FUNCTION_BLOCK FB_VisionStation IMPLEMENTS I_ProcessEquipment
VAR
    // Commissioning FAIL/fault injection; a real camera FAIL cannot be overridden.
    // FALSE = use the real camera verdicts (default)
    // TRUE  = inject FAIL after valid camera evaluation
    bSimulatedFail              : BOOL := FALSE;
    bSimulatedFault             : BOOL := FALSE;

    bEnableInternal             : BOOL;
    bCommissionedInternal       : BOOL;
    bSafetyOkInternal           : BOOL;
    bSupervisionEnableInternal  : BOOL;

    // Nest support and intermediate stop removed from the mechanical design.


    // Vision / flipping tooling feedback.
    bHorizontalBackInternal     : BOOL;
    bHorizontalFrontInternal    : BOOL;
    bVerticalUpInternal         : BOOL;
    bVerticalDownInternal       : BOOL;

    bGripOpenedInternal         : BOOL;
    bGripClosedInternal         : BOOL;
    bRotate0Internal            : BOOL;
    bRotate180Internal          : BOOL;
    bRotate0RawInternal : BOOL;
    bRotate180RawInternal : BOOL;
    bCameraTriggerAcceptedInternal : BOOL;
    bCameraReadyForFlipInternal : BOOL;
    bUseOptimizedSequenceTimingInternal : BOOL;
    rtRotate0Raw : R_TRIG;
    tonFlipDeparture : TON;
    tFlipDepartureFilter : TIME := T#20MS;
    bFlipCaptureActive : BOOL;
    bFlipCaptureActivePrevious : BOOL;
    bFlipStart0Confirmed : BOOL;
    bFlipLeft0 : BOOL;
    bFlip90Seen : BOOL;
    bFlipTriggerLatched : BOOL;
    bFlipCaptureAccepted : BOOL;
    bFlipCaptureWindowMissed : BOOL;
	// Vision / Camera
	

    eStateInternal              : E_PatchStationState := E_PatchStationState.Disabled;
    usiStepInternal             : USINT := 0;
    bHomeInternal               : BOOL;
    bReadyInternal              : BOOL;
    bBusyInternal               : BOOL;
    bCompleteInternal           : BOOL;
    bFaultInternal              : BOOL;
    sDiagnosticInternal         : STRING(120);

    // Output requests.

    bHorizontalBackRequestInternal  : BOOL;
    bHorizontalFrontRequestInternal : BOOL;
    bVerticalUpRequestInternal      : BOOL;
    bVerticalDownRequestInternal    : BOOL;

    bGripCloseRequestInternal       : BOOL;
    bGripOpenRequestInternal        : BOOL;
    bRotate0RequestInternal         : BOOL;
    bRotate180RequestInternal       : BOOL;
	
	bTriggerRequestInternal			: BOOL;
	bChangeProgramRequestInternal	: BOOL;
	bGetResultsRequestInternal		: BOOL;
	bResetResultsRequestInternal	: BOOL;
	nSetProgramNumberInternal		: UDINT;
	bAcknowledgeResultsInternal		: BOOL;
	
	nCurrentProgramNumberInternal	: UDINT;
	bCameraResultsReadyInternal		: BOOL;
	nVisionResultsInternal			: ST_VisionResults;

    bStopRequestInternal        : BOOL;


    // Commissioning timing.
    tonStepDelay                : TON;
    tonRotate180Hold            : TON;
    tonMoveTimeout              : TON;

    tonToolingSensorConflict    : TON;

	tonChangeProgram			: TON := (PT := T#1S);

    tStepDelay                  : TIME := T#100MS;
    tRotate180Hold              : TIME := T#1S;
    tMoveTimeout                : TIME := T#30S;

    tToolingSensorConflict      : TIME := T#300MS;

	tTakingPictureWHileRotating	: TIME := T#100MS; // Delay AFTER the latched 90-degree marker; commission for the desired image.
	tDelayInspectionPlaceHolder	: TIME;

    bStepTargetReached          : BOOL;
    bToolingSensorConflict      : BOOL;
	
	rTrigger						: R_TRIG;
	tonCamera110Rearm             : TON;
	tonCameraTriggerDelay			: ARRAY [1..2] OF TON;
	tonTakingPictureWHileRotating	: TON;
	tonDelayInspectionPlaceHolder	: TON;

    stEmptyVisionResults        : ST_VisionResults;
    stResultInternal            : ST_ProcessResult;
    stProcessSettingsInternal : ST_CameraProcessSettings;
END_VAR

METHOD PUBLIC Cyclic
VAR_INPUT
END_VAR
VAR
	
	

END_VAR
tTakingPictureWHileRotating := UDINT_TO_TIME(stProcessSettingsInternal.udiMovingTriggerDelayMs);
// Marker tracking uses raw feedback; endpoint qualification is independent.
rtRotate0Raw(CLK := bRotate0RawInternal);
bFlipCaptureActive := bEnableInternal AND bCommissionedInternal AND bSafetyOkInternal
    AND NOT bStopRequestInternal
    AND (eStateInternal = E_PatchStationState.Processing) AND (usiStepInternal = 100);
IF NOT bFlipCaptureActive THEN
    bFlipStart0Confirmed := FALSE;
    bFlipLeft0 := FALSE;
    bFlip90Seen := FALSE;
    bFlipTriggerLatched := FALSE;
    bFlipCaptureAccepted := FALSE;
    bFlipCaptureWindowMissed := FALSE;
ELSIF NOT bFlipCaptureActivePrevious THEN
    bFlipStart0Confirmed := bRotate0Internal AND NOT bRotate180RawInternal;
    bFlipLeft0 := FALSE;
    bFlip90Seen := FALSE;
    bFlipTriggerLatched := FALSE;
    bFlipCaptureAccepted := FALSE;
    bFlipCaptureWindowMissed := NOT bFlipStart0Confirmed;
END_IF
tonFlipDeparture(IN := bFlipCaptureActive AND bFlipStart0Confirmed AND NOT bFlipLeft0
    AND NOT bRotate0RawInternal AND NOT bRotate180RawInternal, PT := tFlipDepartureFilter);
IF tonFlipDeparture.Q THEN bFlipLeft0 := TRUE; END_IF
IF bFlipCaptureActive AND bFlipLeft0 AND rtRotate0Raw.Q
    AND NOT bFlip90Seen AND NOT bRotate180RawInternal THEN
    bFlip90Seen := TRUE;
END_IF
tonTakingPictureWHileRotating(IN := bFlipCaptureActive AND bFlip90Seen,
    PT := tTakingPictureWHileRotating);
IF bFlipCaptureActive THEN
    IF bFlipTriggerLatched AND bCameraTriggerAcceptedInternal THEN bFlipCaptureAccepted := TRUE; END_IF
    IF bRotate180RawInternal AND NOT bFlipCaptureAccepted THEN
        bFlipCaptureWindowMissed := TRUE;
    ELSIF tonTakingPictureWHileRotating.Q AND NOT bFlipTriggerLatched
        AND NOT bFlipCaptureWindowMissed THEN
        IF nCurrentProgramNumberInternal = 1 THEN
            bFlipTriggerLatched := TRUE;
        ELSE
            bFlipCaptureWindowMissed := TRUE;
        END_IF
    END_IF
END_IF
bFlipCaptureActivePrevious := bFlipCaptureActive;

// Rearm inspection 2 after entry and confirmed program selection.
tonCamera110Rearm(
    IN := (eStateInternal = E_PatchStationState.Processing)
        AND (usiStepInternal = 110)
        AND (nCurrentProgramNumberInternal = 2)
        AND NOT tonCameraTriggerDelay[1].IN
        AND NOT tonCameraTriggerDelay[2].IN,
    PT := T#500MS
);

bTriggerRequestInternal :=
    (eStateInternal = E_PatchStationState.Processing)
    AND (
        ((usiStepInternal = 100) AND (nCurrentProgramNumberInternal = 1)
            AND bFlipTriggerLatched AND NOT bFlipCaptureWindowMissed)
        OR ((usiStepInternal = 10) AND (nCurrentProgramNumberInternal = 0)
            AND NOT tonCameraTriggerDelay[2].IN)
        OR ((usiStepInternal = 110) AND tonCamera110Rearm.Q)
        OR ((usiStepInternal = 180) AND (nCurrentProgramNumberInternal = 3))
    );
bGetResultsRequestInternal := FALSE;
bAcknowledgeResultsInternal := FALSE;
bChangeProgramRequestInternal := FALSE;
tonCameraTriggerDelay[1](PT := T#500MS);
// Keep the program 0-to-1 timer running while pick and mounting proceed.
IF (eStateInternal = E_PatchStationState.Processing)
    AND ((usiStepInternal = 10) OR (bUseOptimizedSequenceTimingInternal AND (usiStepInternal <= 90))) THEN
    tonCameraTriggerDelay[2](PT := T#200MS);
ELSE
    tonCameraTriggerDelay[2](PT := T#500MS);
END_IF
tonDelayInspectionPlaceHolder(PT := tDelayInspectionPlaceHolder);

 // ============================================================================
 // Vision Station / Flipping sequence
 // ============================================================================
 // Home:
 //
 // Process (active mechanical steps and camera inspections):
 //
 //   10  1st Vision Inspection - Program 0
 //   30  Vertical FULL DOWN - pick
 //   40  Grip CLOSE
 //   50  Vertical UP
 //   60  Horizontal FRONT
 //   80  Vertical UP before flip
 //   100  Rotate 180; timed Program 1 capture and result acquisition
 //   110  3rd Vision Inspection - Program 2
 //  150  Grip OPEN - release part
 //  160  Vertical UP after release
 //  170  Return tooling HOME
 //  180  4th Vision Inspection - Program 3
 //  190  Aggregate four camera verdicts, then Complete


// ============================================================================
// DEFAULT REQUESTS
// ============================================================================

// Default all requests OFF. Each active state below explicitly builds the
// desired command state and never energises opposing coils simultaneously.

bHorizontalBackRequestInternal := FALSE;
bHorizontalFrontRequestInternal := FALSE;
bVerticalUpRequestInternal := FALSE;
bVerticalDownRequestInternal := FALSE;

bGripCloseRequestInternal := FALSE;
bGripOpenRequestInternal := FALSE;
bRotate0RequestInternal := FALSE;
bRotate180RequestInternal := FALSE;

//bStepTargetReached := FALSE;
bFaultInternal := FALSE;


// ============================================================================
// HOME FEEDBACK
// ============================================================================

bHomeInternal :=
    bHorizontalBackInternal AND NOT bHorizontalFrontInternal
    AND bVerticalUpInternal AND NOT bVerticalDownInternal
    AND bGripOpenedInternal AND NOT bGripClosedInternal
    AND bRotate0Internal AND NOT bRotate180Internal;


// ============================================================================
// TOOLING SENSOR PLAUSIBILITY
// ============================================================================

bToolingSensorConflict :=
    (bHorizontalBackInternal AND bHorizontalFrontInternal)
    OR (bVerticalUpInternal AND bVerticalDownInternal)
    OR (bGripOpenedInternal AND bGripClosedInternal)
    OR (bRotate0RawInternal AND bRotate180RawInternal);

// End-position sensors can overlap briefly during pneumatic transitions.
// Only treat contradictory feedback as a real fault when it persists.
tonToolingSensorConflict(
    IN := bSupervisionEnableInternal
        AND bSafetyOkInternal
        AND bToolingSensorConflict,
    PT := tToolingSensorConflict
);


// ============================================================================
// MAIN STATE CONTROL
// ============================================================================

IF bEnableInternal AND bSimulatedFault THEN

    eStateInternal := E_PatchStationState.Fault;
    usiStepInternal := 0;
    sDiagnosticInternal := 'Vision: simulated station fault';


ELSIF bFlipCaptureWindowMissed THEN
    eStateInternal := E_PatchStationState.Fault;
    usiStepInternal := 0;
    bTriggerRequestInternal := FALSE;
    sDiagnosticInternal := 'Vision: rotation reference or moving-image window missed';
    stResultInternal.bValid := TRUE;
    stResultInternal.bPassed := FALSE;
    stResultInternal.eCode := E_ProcessResultCode.Fail;
    stResultInternal.udiFaultCode := 12;
    stResultInternal.udiAlertCode := 0;
    stResultInternal.sDetail := sDiagnosticInternal;

ELSIF tonToolingSensorConflict.Q THEN

    eStateInternal := E_PatchStationState.Fault;
    usiStepInternal := 0;
    sDiagnosticInternal := 'Vision: contradictory tooling sensors';


ELSIF bFaultInternal THEN

    // Fault state handled below.


ELSIF bStopRequestInternal THEN

    // Controlled station stop: start one deterministic return-to-home sequence.
    // Clear the request here so the homing step counter is not reset every scan.
    eStateInternal := E_PatchStationState.Homing;
    usiStepInternal := 0;
    bStopRequestInternal := FALSE;


ELSIF NOT bCommissionedInternal THEN

    eStateInternal := E_PatchStationState.Disabled;
    usiStepInternal := 0;
    sDiagnosticInternal := 'Vision: station disabled';


ELSIF NOT bSafetyOkInternal THEN

    eStateInternal := E_PatchStationState.Disabled;
    usiStepInternal := 0;
    sDiagnosticInternal := 'Vision: disabled by Safety';


ELSIF NOT bEnableInternal THEN

    IF bHomeInternal THEN

        eStateInternal := E_PatchStationState.Disabled;
        usiStepInternal := 0;
        sDiagnosticInternal := 'Vision: disabled - tooling home';

    ELSE

        eStateInternal := E_PatchStationState.Homing;
        usiStepInternal := 0;
        sDiagnosticInternal := 'Vision: disabled - returning tooling home';

    END_IF


ELSE

    CASE eStateInternal OF


        // ====================================================================
        // DISABLED / HOMING
        // ====================================================================

        E_PatchStationState.Disabled,
        E_PatchStationState.Homing:

            // Deterministic / collision-conscious home sequence used by
            // System Initialising and controlled station recovery.
            //
			// Defined HOME:

            // Request program 0 during homing; mechanical Ready still does not confirm camera Ready.
            
			//Leaving camera with the right program to performance first test--------------------------
			
			IF nCurrentProgramNumberInternal<> 0 THEN
				
				nSetProgramNumberInternal				:= 0;
				bChangeProgramRequestInternal			:= TRUE;
				
			ELSIF nCurrentProgramNumberInternal = 0 THEN
				
				bChangeProgramRequestInternal			:= FALSE;
				
			END_IF
			

            
			//-------------------------------------------------------------------------------------------
            IF usiStepInternal = 0 THEN

                IF bHomeInternal THEN
                    usiStepInternal := 70;
                ELSE
                    usiStepInternal := 10;
                END_IF

            END_IF


            CASE usiStepInternal OF
			

				10: // Vertical UP

                    bVerticalUpRequestInternal := NOT bVerticalUpInternal;

                    bStepTargetReached :=
                        bVerticalUpInternal
                        AND NOT bVerticalDownInternal;

                    sDiagnosticInternal := 'Vision homing: vertical UP';


                30: // Rotate gripper to 0 deg

                    bVerticalUpRequestInternal := NOT bVerticalUpInternal;

                    bRotate0RequestInternal := NOT bRotate0Internal;

                    bStepTargetReached :=
                        bRotate0Internal
                        AND NOT bRotate180Internal;

                    sDiagnosticInternal := 'Vision homing: rotate grip to 0 deg';


                40: // Grip OPEN

                    bVerticalUpRequestInternal := NOT bVerticalUpInternal;

                    bRotate0RequestInternal := NOT bRotate0Internal;
                    bGripOpenRequestInternal := NOT bGripOpenedInternal;

                    bStepTargetReached :=
                        bGripOpenedInternal
                        AND NOT bGripClosedInternal;

                    sDiagnosticInternal := 'Vision homing: grip OPEN';


                60: // Horizontal slide BACK

                    bVerticalUpRequestInternal := NOT bVerticalUpInternal;

                    bRotate0RequestInternal := NOT bRotate0Internal;
                    bGripOpenRequestInternal := NOT bGripOpenedInternal;



                    bHorizontalBackRequestInternal := NOT bHorizontalBackInternal;

                    bStepTargetReached :=
                        bHorizontalBackInternal
                        AND NOT bHorizontalFrontInternal;

                    sDiagnosticInternal := 'Vision homing: horizontal slide BACK';


                70: // Verify complete HOME before declaring Ready

                    bHorizontalBackRequestInternal := NOT bHorizontalBackInternal;
                    bVerticalUpRequestInternal := NOT bVerticalUpInternal;



                    bGripOpenRequestInternal := NOT bGripOpenedInternal;
                    bRotate0RequestInternal := NOT bRotate0Internal;

                    // Modified by Thays - TEMPORARY: verify mechanical HOME without requiring Keyence program 0.
                    // bStepTargetReached := bHomeInternal AND (nCurrentProgramNumberInternal = 0);
                    bStepTargetReached := bHomeInternal;

                    sDiagnosticInternal := 'Vision homing: verifying HOME';
					

                ELSE

                    usiStepInternal := 10;
                    bStepTargetReached := FALSE;

            END_CASE


            tonStepDelay(
                IN := bStepTargetReached,
                PT := tStepDelay
            );

            tonMoveTimeout(
                IN := NOT bStepTargetReached,
                PT := tMoveTimeout
            );


            // ================================================================
            // HOMING TIMEOUT SUPERVISION
            // ================================================================

            IF tonMoveTimeout.Q THEN

                tonMoveTimeout(IN := FALSE);
                tonStepDelay(IN := FALSE);

                eStateInternal := E_PatchStationState.Fault;
                usiStepInternal := 0;

                sDiagnosticInternal := 'Vision: homing movement timeout';

                stResultInternal.bValid := TRUE;
                stResultInternal.bPassed := FALSE;
                stResultInternal.eCode := E_ProcessResultCode.Fail;
                stResultInternal.udiFaultCode := 11;
                stResultInternal.udiAlertCode := 0;
                stResultInternal.sDetail := 'Vision homing movement timeout';


            ELSIF tonStepDelay.Q THEN

                tonMoveTimeout(IN := FALSE);
                tonStepDelay(IN := FALSE);

                IF usiStepInternal < 70 THEN

                    IF usiStepInternal = 10 THEN
                        usiStepInternal := 30;
                    ELSIF usiStepInternal = 40 THEN
                        usiStepInternal := 60;
                    ELSE
                        usiStepInternal := usiStepInternal + 10;
                    END_IF

                ELSE

                    eStateInternal := E_PatchStationState.Ready;
                    usiStepInternal := 0;
                    sDiagnosticInternal := 'Vision: ready - tooling home';
					bStepTargetReached					:= FALSE;

                END_IF

            END_IF


        // ====================================================================
        // READY
        // ====================================================================

        E_PatchStationState.Ready:

            // Reset can enter Ready directly when tooling is already home.
            // Restore the camera independently of the mechanical homing path.
            IF nCurrentProgramNumberInternal <> 0 THEN
                nSetProgramNumberInternal := 0;
                bChangeProgramRequestInternal := TRUE;
            END_IF

            tonStepDelay(IN := FALSE);
            tonRotate180Hold(IN := FALSE);
            tonMoveTimeout(IN := FALSE);

            // Hold/restore the defined HOME position.

            bHorizontalBackRequestInternal := NOT bHorizontalBackInternal;
            bVerticalUpRequestInternal := NOT bVerticalUpInternal;



            bGripOpenRequestInternal := NOT bGripOpenedInternal;
            bRotate0RequestInternal := NOT bRotate0Internal;

            IF NOT bHomeInternal THEN

                eStateInternal := E_PatchStationState.Homing;
                sDiagnosticInternal := 'Vision: lost home - recovering';

            ELSE

                sDiagnosticInternal := 'Vision: ready - waiting for cycle start';

            END_IF


        // ====================================================================
        // PROCESSING
        // ====================================================================

        E_PatchStationState.Processing:

            // Each scan must prove completion of the active step.
            bStepTargetReached := FALSE;

            // Continue the first camera handshake while automatic tooling moves.
            IF (usiStepInternal = 10) OR (bUseOptimizedSequenceTimingInternal AND (usiStepInternal <= 90)) THEN
                IF tonCameraTriggerDelay[1].Q THEN
                    tonCameraTriggerDelay[1].IN := FALSE;
                    tonCameraTriggerDelay[2].IN := TRUE;
                END_IF

                IF tonCameraTriggerDelay[2].IN THEN
                    nSetProgramNumberInternal := 1;
                    bChangeProgramRequestInternal := (nCurrentProgramNumberInternal <> 1);
                ELSIF (usiStepInternal = 10) AND (nCurrentProgramNumberInternal = 0)
                    AND bCameraResultsReadyInternal THEN
                    bGetResultsRequestInternal := TRUE;
                    bAcknowledgeResultsInternal := TRUE;
                    tonCameraTriggerDelay[1].IN := TRUE;
                ELSIF (usiStepInternal = 10) AND NOT tonCameraTriggerDelay[1].IN
                    AND (nCurrentProgramNumberInternal <> 0) THEN
                    nSetProgramNumberInternal := 0;
                    bChangeProgramRequestInternal := TRUE;
                END_IF
            END_IF

            CASE usiStepInternal OF

                10: // Keep the part stationary until the first result has been copied.
                    bStepTargetReached := nVisionResultsInternal.aInspectionCompleted[1]
                        AND (tonCameraTriggerDelay[1].IN OR tonCameraTriggerDelay[2].IN)
                        AND (bUseOptimizedSequenceTimingInternal
                            OR (tonCameraTriggerDelay[2].Q AND (nCurrentProgramNumberInternal = 1)));
                    sDiagnosticInternal := 'Vision: Camera first inspection';

                20: // Prepare existing tooling for pick.
                    bHorizontalBackRequestInternal := NOT bHorizontalBackInternal;
                    bVerticalUpRequestInternal := NOT bVerticalUpInternal;
                    bGripOpenRequestInternal := NOT bGripOpenedInternal;
                    bRotate0RequestInternal := NOT bRotate0Internal;
                    bStepTargetReached := bHorizontalBackInternal AND NOT bHorizontalFrontInternal
                        AND bVerticalUpInternal AND NOT bVerticalDownInternal
                        AND bGripOpenedInternal AND NOT bGripClosedInternal
                        AND bRotate0Internal AND NOT bRotate180Internal;
                    sDiagnosticInternal := 'Vision: preparing pick tooling';

                30:

                    bHorizontalBackRequestInternal := NOT bHorizontalBackInternal;

                    // Coil5 = OFF.


                    bVerticalDownRequestInternal := NOT bVerticalDownInternal;

                    bGripOpenRequestInternal := NOT bGripOpenedInternal;
                    bRotate0RequestInternal := NOT bRotate0Internal;

                    bStepTargetReached :=
                        bVerticalDownInternal
                        AND NOT bVerticalUpInternal;

                    sDiagnosticInternal := 'Vision: vertical FULL DOWN - pick';


                // ------------------------------------------------------------
                // STEP 40 - GRIP CLOSE AT FULL DOWN
                // ------------------------------------------------------------

                40:

                    bHorizontalBackRequestInternal := NOT bHorizontalBackInternal;

                    // Keep stop retracted while gripping at FULL DOWN.


                    bVerticalDownRequestInternal := NOT bVerticalDownInternal;

                    bGripCloseRequestInternal := NOT bGripClosedInternal;
                    bRotate0RequestInternal := NOT bRotate0Internal;

                    bStepTargetReached :=
                        bGripClosedInternal
                        AND NOT bGripOpenedInternal;

                    sDiagnosticInternal := 'Vision: grip CLOSE at full DOWN';


                // ------------------------------------------------------------
                // STEP 50 - VERTICAL UP
                // ------------------------------------------------------------

                50:

                    bHorizontalBackRequestInternal := NOT bHorizontalBackInternal;
                    bVerticalUpRequestInternal := NOT bVerticalUpInternal;

                    // Keep stop retracted until vertical is safely UP.


                    bGripCloseRequestInternal := NOT bGripClosedInternal;
                    bRotate0RequestInternal := NOT bRotate0Internal;

                    bStepTargetReached :=
                        bVerticalUpInternal
                        AND NOT bVerticalDownInternal;

                    sDiagnosticInternal := 'Vision: vertical UP with part';


                // ------------------------------------------------------------
                // STEP 60 - HORIZONTAL FRONT
                // ------------------------------------------------------------

                60:

                    bHorizontalFrontRequestInternal := NOT bHorizontalFrontInternal;
                    bVerticalUpRequestInternal := NOT bVerticalUpInternal;

                    // before commanding the next DOWN movement.


                    bGripCloseRequestInternal := NOT bGripClosedInternal;
                    bRotate0RequestInternal := NOT bRotate0Internal;

                    bStepTargetReached :=
                        bHorizontalFrontInternal
                        AND NOT bHorizontalBackInternal;

                    sDiagnosticInternal := 'Vision: horizontal FRONT';


                // ------------------------------------------------------------
                // ------------------------------------------------------------

                70: // Two-position vertical cylinder: use actual DOWN feedback.
                    bHorizontalFrontRequestInternal := NOT bHorizontalFrontInternal;
                    bVerticalDownRequestInternal := NOT bVerticalDownInternal;
                    bGripCloseRequestInternal := NOT bGripClosedInternal;
                    bRotate0RequestInternal := NOT bRotate0Internal;
                    bStepTargetReached := bVerticalDownInternal AND NOT bVerticalUpInternal;
                    IF bStepTargetReached THEN
                        sDiagnosticInternal := 'Vision: PBUP mounting - holding DOWN for 1 s';
                    ELSE
                        sDiagnosticInternal := 'Vision: vertical DOWN - front position';
                    END_IF

                80:

                    bHorizontalFrontRequestInternal := NOT bHorizontalFrontInternal;
                    bVerticalUpRequestInternal := NOT bVerticalUpInternal;



                    bGripCloseRequestInternal := NOT bGripClosedInternal;
                    bRotate0RequestInternal := NOT bRotate0Internal;

                    // FIX: removed simultaneous retract request from Step 70.
                    // OLD: bStepTargetReached :=
                    //          (bVerticalUpInternal AND NOT bVerticalDownInternal)
                    bStepTargetReached :=
                        bVerticalUpInternal
                        AND NOT bVerticalDownInternal;

                    sDiagnosticInternal := 'Vision: vertical UP before flip';

                // ------------------------------------------------------------
                // ------------------------------------------------------------

                90: // Verify clearance before rotation; no nest support is fitted.
                    bHorizontalFrontRequestInternal := NOT bHorizontalFrontInternal;
                    bVerticalUpRequestInternal := NOT bVerticalUpInternal;
                    bGripCloseRequestInternal := NOT bGripClosedInternal;
                    bRotate0RequestInternal := NOT bRotate0Internal;
                    bStepTargetReached := bVerticalUpInternal AND NOT bVerticalDownInternal
                        AND bRotate0Internal AND NOT bRotate180Internal;
                    IF bUseOptimizedSequenceTimingInternal
                        AND NOT (tonCameraTriggerDelay[2].Q AND (nCurrentProgramNumberInternal = 1)
                            AND bCameraReadyForFlipInternal) THEN
                        bStepTargetReached := FALSE;
                        sDiagnosticInternal := 'Vision: waiting for camera program 1 ready';
                    ELSE
                        sDiagnosticInternal := 'Vision: verify UP before flip';
                    END_IF

                100: // Support retraction was confirmed in step 90.

					// Program 1 trigger now follows the first valid 90-degree marker.

                    bHorizontalFrontRequestInternal := NOT bHorizontalFrontInternal;
                    bVerticalUpRequestInternal := NOT bVerticalUpInternal;


                    bGripCloseRequestInternal := NOT bGripClosedInternal;
                    bRotate180RequestInternal := NOT bRotate180Internal;

                    // Acquire program 1 before requesting program 2.
                    
					//Camera
					IF nCurrentProgramNumberInternal = 1 THEN
					
					IF bCameraResultsReadyInternal AND NOT tonCameraTriggerDelay[2].IN THEN
						
						bGetResultsRequestInternal			:= TRUE;
						bAcknowledgeResultsInternal			:= TRUE;
						tonCameraTriggerDelay[1].IN			:= TRUE;
						
						
					END_IF
					
					END_IF
					IF tonCameraTriggerDelay[1].Q THEN
							
							bGetResultsRequestInternal			:= FALSE;
							bAcknowledgeResultsInternal			:= FALSE;
							nSetProgramNumberInternal			:= 2;
							tonDelayInspectionPlaceHolder.IN	:= TRUE;
							bChangeProgramRequestInternal		:= TRUE;
							tonCameraTriggerDelay[2].IN			:= TRUE;
							tonCameraTriggerDelay[1].IN			:= FALSE;
							
							
					END_IF
					// Hold program selection until the camera reports the requested program.
                    IF tonCameraTriggerDelay[2].IN THEN
                        nSetProgramNumberInternal := 2;
                        bChangeProgramRequestInternal := (nCurrentProgramNumberInternal <> 2);
                    END_IF
                    IF tonCameraTriggerDelay[2].Q AND (nCurrentProgramNumberInternal = 2) THEN
							
							
							bChangeProgramRequestInternal		:= FALSE;

							
							
					END_IF
					// The moving-image delay is not restarted by the program-change placeholder.
					
					bStepTargetReached := tonDelayInspectionPlaceHolder.Q
                        AND (nCurrentProgramNumberInternal = 2)
                        AND bRotate180Internal AND NOT bRotate0Internal;
					
					                    
                    // Physical 180 completion is now qualified above before inspection 3.
                    //tonDelayInspectionPlaceHolder.IN := bRotate180Internal AND NOT bRotate0Internal;
                    //bStepTargetReached := bRotate180Internal AND NOT bRotate0Internal AND tonDelayInspectionPlaceHolder.Q;
                    sDiagnosticInternal := 'Vision: rotate 180, marker-based image 2';
				
                // Pending: accepted-trigger/fresh-result handshake and supervised visual inspection recovery.
        
				// ------------------------------------------------------------
                // STEP 110 - CAMERA PROGRAM 2 - THIRD INSPECTION
                // ------------------------------------------------------------
				
				110:
					tonDelayInspectionPlaceHolder.IN		:= FALSE;

                    // Acquire program 2 before requesting program 3.
                    
					IF nCurrentProgramNumberInternal = 2 THEN
					
					IF bCameraResultsReadyInternal AND NOT tonCameraTriggerDelay[2].IN THEN
						
						bGetResultsRequestInternal			:= TRUE;
						bAcknowledgeResultsInternal			:= TRUE;
						tonCameraTriggerDelay[1].IN			:= TRUE;
						
						
					END_IF
					END_IF
					
					IF tonCameraTriggerDelay[1].Q THEN
							
							bGetResultsRequestInternal			:= FALSE;
							bAcknowledgeResultsInternal			:= FALSE;
							nSetProgramNumberInternal			:= 3;
							bChangeProgramRequestInternal		:= TRUE;
							tonCameraTriggerDelay[2].IN			:= TRUE;
							tonCameraTriggerDelay[1].IN			:= FALSE;
							
							
					END_IF
					// Hold program selection until the camera reports the requested program.
                    IF tonCameraTriggerDelay[2].IN THEN
                        nSetProgramNumberInternal := 3;
                        bChangeProgramRequestInternal := (nCurrentProgramNumberInternal <> 3);
                    END_IF
                    IF tonCameraTriggerDelay[2].Q AND (nCurrentProgramNumberInternal = 3) THEN
							
							
							bChangeProgramRequestInternal		:= FALSE;
							bStepTargetReached					:= TRUE;
                            // Keep delay 2 complete until this step advances.
							
							
					END_IF
				
                    
                    //bStepTargetReached := TRUE; // Modified by Thays - no camera inspection result.

                // ------------------------------------------------------------
                // STEP 120 - ROTATE BACK TO 0
                // ------------------------------------------------------------

                120: 

                    bHorizontalFrontRequestInternal := NOT bHorizontalFrontInternal;
                    bVerticalUpRequestInternal := NOT bVerticalUpInternal;


                    bGripCloseRequestInternal := NOT bGripClosedInternal;
                    bRotate0RequestInternal := NOT bRotate0Internal;

                    // simultaneously while rotating, conflicting with rotation permissive.
                    // OLD: bStepTargetReached :=
                    //          (bRotate0Internal AND NOT bRotate180Internal)
                    //          (*AND bGetResultsReadyRequestInternal*);
                    bStepTargetReached :=
                        bRotate0Internal
                        AND NOT bRotate180Internal;

                    sDiagnosticInternal := 'Vision: rotate back to 0';

                // ------------------------------------------------------------
                // ------------------------------------------------------------
				
				
					

                130: // Verify tooling after rotation before replace.
                    bHorizontalFrontRequestInternal := NOT bHorizontalFrontInternal;
                    bVerticalUpRequestInternal := NOT bVerticalUpInternal;
                    bGripCloseRequestInternal := NOT bGripClosedInternal;
                    bStepTargetReached := bHorizontalFrontInternal AND NOT bHorizontalBackInternal
                        AND bVerticalUpInternal AND NOT bVerticalDownInternal
                        AND bGripClosedInternal AND NOT bGripOpenedInternal
                        AND bRotate0Internal AND NOT bRotate180Internal;
                    sDiagnosticInternal := 'Vision: preparing replace tooling';

                140: // Two-position vertical cylinder: use actual DOWN feedback.
                    bHorizontalFrontRequestInternal := NOT bHorizontalFrontInternal;
                    bVerticalDownRequestInternal := NOT bVerticalDownInternal;
                    bGripCloseRequestInternal := NOT bGripClosedInternal;
                    bRotate0RequestInternal := NOT bRotate0Internal;
                    bStepTargetReached := bVerticalDownInternal AND NOT bVerticalUpInternal;
                    sDiagnosticInternal := 'Vision: vertical DOWN - replace part';

                150: // Release only at the confirmed DOWN endpoint.
                    bHorizontalFrontRequestInternal := NOT bHorizontalFrontInternal;
                    bVerticalDownRequestInternal := NOT bVerticalDownInternal;
                    bGripOpenRequestInternal := bVerticalDownInternal AND NOT bVerticalUpInternal
                        AND NOT bGripOpenedInternal;
                    bRotate0RequestInternal := NOT bRotate0Internal;
                    bStepTargetReached := bVerticalDownInternal AND NOT bVerticalUpInternal
                        AND bGripOpenedInternal AND NOT bGripClosedInternal;
                    sDiagnosticInternal := 'Vision: grip OPEN at DOWN - release part';

                160: // FIX: renumbered after separating support movements.

                    bHorizontalFrontRequestInternal := NOT bHorizontalFrontInternal;

                    bVerticalUpRequestInternal := NOT bVerticalUpInternal;


                    bGripOpenRequestInternal := NOT bGripOpenedInternal;
                    bRotate0RequestInternal := NOT bRotate0Internal;

                    bStepTargetReached :=
                        bVerticalUpInternal
                        AND NOT bVerticalDownInternal;

                    sDiagnosticInternal := 'Vision: vertical UP after release';


                // ------------------------------------------------------------
                // STEP 170 - RETURN HOME
                // ------------------------------------------------------------

                170: // FIX: renumbered after separating support movements.

                    bHorizontalBackRequestInternal := NOT bHorizontalBackInternal;
                    bVerticalUpRequestInternal := NOT bVerticalUpInternal;




                    bGripOpenRequestInternal := NOT bGripOpenedInternal;
                    bRotate0RequestInternal := NOT bRotate0Internal;

                    bStepTargetReached := bHomeInternal;

                    sDiagnosticInternal := 'Vision: returning tooling to home';
				
				// ------------------------------------------------------------
                // STEP 180 - CAMERA PBUB - FOURTH INSPECTION
                // ------------------------------------------------------------                
                180:
                    // Only program 3 may supply this inspection's result.
                    IF (nCurrentProgramNumberInternal = 3)
                        AND bCameraResultsReadyInternal
                        AND NOT tonCameraTriggerDelay[2].IN
                    THEN
                        bGetResultsRequestInternal := TRUE;
                        bAcknowledgeResultsInternal := TRUE;
                        tonCameraTriggerDelay[1].IN := TRUE;
                    END_IF

                    // Finish the delay even after the camera returns to program 0.
                    IF tonCameraTriggerDelay[1].Q THEN
                        bGetResultsRequestInternal := FALSE;
                        bAcknowledgeResultsInternal := FALSE;
                        nSetProgramNumberInternal := 0;
                        bChangeProgramRequestInternal := TRUE;
                        tonCameraTriggerDelay[2].IN := TRUE;
                        tonCameraTriggerDelay[1].IN := FALSE;
                    END_IF

                    // Hold program selection until the camera reports the requested program.
                    IF tonCameraTriggerDelay[2].IN THEN
                        nSetProgramNumberInternal := 0;
                        bChangeProgramRequestInternal := (nCurrentProgramNumberInternal <> 0);
                    END_IF
                    IF tonCameraTriggerDelay[2].Q AND (nCurrentProgramNumberInternal = 0) THEN
                        bChangeProgramRequestInternal := FALSE;
                        bStepTargetReached := TRUE;
                        // Keep delay 2 complete until this step advances.
                    END_IF

                    sDiagnosticInternal := 'Vision: Camera fourth inspection';

				190:
				
					bStepTargetReached := TRUE;

                // Pending: accepted-trigger/fresh-result handshake and supervised visual inspection recovery.

                ELSE

                    eStateInternal := E_PatchStationState.Fault;
                    usiStepInternal := 0;
                    sDiagnosticInternal := 'Vision: invalid sequence step';

            END_CASE


            // ================================================================
            // PROCESSING TRANSITIONS
            // ================================================================

            
                // PBUP mounting: require continuous DOWN confirmation for 1 s.
                // Existing transition/reset logic rearms this timer for each step.
                IF usiStepInternal = 70 THEN
                    tonStepDelay(
                        IN := bStepTargetReached,
                        PT := T#1S
                    );
                ELSE
                    tonStepDelay(
                        IN := bStepTargetReached,
                        PT := tStepDelay
                    );
                END_IF



            tonMoveTimeout(
                IN := NOT bStepTargetReached,
                PT := tMoveTimeout
            );


            // ================================================================
            // PROCESSING MOVEMENT TIMEOUT SUPERVISION
            // ================================================================

            IF tonMoveTimeout.Q THEN

                tonMoveTimeout(IN := FALSE);
                tonStepDelay(IN := FALSE);
                tonRotate180Hold(IN := FALSE);

                eStateInternal := E_PatchStationState.Fault;
                usiStepInternal := 0;

                bChangeProgramRequestInternal := FALSE;
                bGetResultsRequestInternal := FALSE;
                bAcknowledgeResultsInternal := FALSE;

                sDiagnosticInternal := 'Vision: tooling movement or camera handshake timeout';

                stResultInternal.bValid := TRUE;
                stResultInternal.bPassed := FALSE;
                stResultInternal.eCode := E_ProcessResultCode.Fail;
                stResultInternal.udiFaultCode := 10;
                stResultInternal.udiAlertCode := 0;
                stResultInternal.sDetail := sDiagnosticInternal;

			(*
            ELSIF (usiStepInternal = 20) AND bStepTargetReached THEN

                tonMoveTimeout(IN := FALSE);
                tonRotate180Hold(IN := FALSE);
                // FIX CAMERA PREPARATION: route through camera 2 placeholder.
                // OLD: usiStepInternal := 100;
                usiStepInternal := 95;*)


            ELSIF (usiStepInternal < 190) AND tonStepDelay.Q THEN

                tonMoveTimeout(IN := FALSE);
                tonStepDelay(IN := FALSE);

                // Advance through the active steps in increments of 10.
              
                // Keep the first camera handshake through step 90.
                IF NOT bUseOptimizedSequenceTimingInternal OR (usiStepInternal >= 90) THEN
                    tonCameraTriggerDelay[1](IN := FALSE);
                    tonCameraTriggerDelay[2](IN := FALSE);
                END_IF
                usiStepInternal := usiStepInternal + 10;
            ELSIF usiStepInternal = 190 THEN

                    stResultInternal.CameraResults := nVisionResultsInternal;
                    stResultInternal.udiFaultCode := 0;
                    stResultInternal.udiAlertCode := 0;
                    stResultInternal.bValid :=
                        nVisionResultsInternal.aInspectionCompleted[1]
                        AND nVisionResultsInternal.aInspectionCompleted[2]
                        AND nVisionResultsInternal.aInspectionCompleted[3]
                        AND nVisionResultsInternal.aInspectionCompleted[4];

                    IF stResultInternal.bValid THEN
                        stResultInternal.bPassed :=
                            nVisionResultsInternal.aInspectionPassed[1]
                            AND nVisionResultsInternal.aInspectionPassed[2]
                            AND nVisionResultsInternal.aInspectionPassed[3]
                            AND nVisionResultsInternal.aInspectionPassed[4]
                            AND NOT bSimulatedFail;
                        stResultInternal.CameraResults.bGeneralPass := stResultInternal.bPassed;
                        stResultInternal.CameraResults.bGeneralFail := NOT stResultInternal.bPassed;

                        IF stResultInternal.bPassed THEN
                            stResultInternal.eCode := E_ProcessResultCode.Pass;
                            stResultInternal.sDetail := 'Vision: four camera inspections PASS';
                        ELSE
                            stResultInternal.eCode := E_ProcessResultCode.Fail;
                            stResultInternal.sDetail := 'Vision: camera inspection FAIL or commissioning FAIL injection';
                        END_IF
                        eStateInternal := E_PatchStationState.Complete;
                    ELSE
                        // No valid automatic verdict: retain the existing fault workflow.
                        stResultInternal.bPassed := FALSE;
                        stResultInternal.eCode := E_ProcessResultCode.None;
                        stResultInternal.udiFaultCode := 11;
                        stResultInternal.sDetail := 'Vision: incomplete camera results - manual inspection required';
                        sDiagnosticInternal := stResultInternal.sDetail;
                        eStateInternal := E_PatchStationState.Fault;
                    END_IF
                    usiStepInternal := 0;

                END_IF

           


        // ====================================================================
        // COMPLETE
        // ====================================================================

        E_PatchStationState.Complete:

            tonStepDelay(IN := FALSE);
            tonRotate180Hold(IN := FALSE);
            tonMoveTimeout(IN := FALSE);

            // Keep/restore HOME after process completion.

            bHorizontalBackRequestInternal := NOT bHorizontalBackInternal;
            bVerticalUpRequestInternal := NOT bVerticalUpInternal;



            bGripOpenRequestInternal := NOT bGripOpenedInternal;
            bRotate0RequestInternal := NOT bRotate0Internal;

            sDiagnosticInternal := 'Vision: flipping complete';


        // ====================================================================
        // FAULT
        // ====================================================================

        E_PatchStationState.Fault:

            tonStepDelay(IN := FALSE);
            tonRotate180Hold(IN := FALSE);
            tonMoveTimeout(IN := FALSE);

            IF stResultInternal.udiFaultCode = 12 THEN
                sDiagnosticInternal := stResultInternal.sDetail;
            ELSE
                sDiagnosticInternal := 'Vision: fault';
            END_IF


        ELSE

            eStateInternal := E_PatchStationState.Fault;
            usiStepInternal := 0;
            sDiagnosticInternal := 'Vision: invalid station state';

    END_CASE

END_IF


// ============================================================================
// FINAL MECHANICAL MOVEMENT INTERLOCKS
// ============================================================================
//
// Independent mechanical permissives applied AFTER the state machine.
// These prevent unsafe movement requests from reaching the physical outputs
// even if a future sequence modification generates an invalid combination.


// ============================================================================
// HORIZONTAL MOVEMENT PERMISSIVE
// ============================================================================
//
// Horizontal movement is only permitted when the vertical tooling is
// positively confirmed UP.

IF NOT (
    bVerticalUpInternal
    AND NOT bVerticalDownInternal
) THEN

    bHorizontalBackRequestInternal := FALSE;
    bHorizontalFrontRequestInternal := FALSE;

END_IF


// ============================================================================
// ROTATION MOVEMENT PERMISSIVE
// ============================================================================
//
// Rotation is only permitted when:
//   Vertical = UP

IF NOT (
    bVerticalUpInternal
    AND NOT bVerticalDownInternal
) THEN

    bRotate0RequestInternal := FALSE;
    bRotate180RequestInternal := FALSE;

END_IF


// ============================================================================
// OPPOSING OUTPUT HARD INTERLOCKS
// ============================================================================
//
// Never allow opposing pneumatic requests simultaneously.
// If both commands are requested, remove BOTH requests.
// Existing timeout supervision will detect failure to reach the target.


// Horizontal Back / Front
IF bHorizontalBackRequestInternal
    AND bHorizontalFrontRequestInternal
THEN

    bHorizontalBackRequestInternal := FALSE;
    bHorizontalFrontRequestInternal := FALSE;

END_IF


// Vertical Up / Down
IF bVerticalUpRequestInternal
    AND bVerticalDownRequestInternal
THEN

    bVerticalUpRequestInternal := FALSE;
    bVerticalDownRequestInternal := FALSE;

END_IF


// Grip Close / Open
IF bGripCloseRequestInternal
    AND bGripOpenRequestInternal
THEN

    bGripCloseRequestInternal := FALSE;
    bGripOpenRequestInternal := FALSE;

END_IF


// Rotation 0 / 180
IF bRotate0RequestInternal
    AND bRotate180RequestInternal
THEN

    bRotate0RequestInternal := FALSE;
    bRotate180RequestInternal := FALSE;

END_IF


// Clear pending camera delays after completion, stop, disable or fault.
IF eStateInternal <> E_PatchStationState.Processing THEN
    tonCameraTriggerDelay[1](IN := FALSE);
    tonCameraTriggerDelay[2](IN := FALSE);
    tonCamera110Rearm(IN := FALSE);
    tonTakingPictureWHileRotating(IN := FALSE);
    tonDelayInspectionPlaceHolder(IN := FALSE);
    bTriggerRequestInternal := FALSE;
END_IF

// ============================================================================
// STATUS
// ============================================================================

bReadyInternal :=
    (eStateInternal = E_PatchStationState.Ready)
    AND bHomeInternal;

bBusyInternal :=
    (eStateInternal = E_PatchStationState.Processing)
    OR ((eStateInternal = E_PatchStationState.Homing) AND NOT bHomeInternal);

bCompleteInternal :=
    (eStateInternal = E_PatchStationState.Complete);

bFaultInternal :=
    (eStateInternal = E_PatchStationState.Fault);
END_METHOD

METHOD PUBLIC GetResult : ST_ProcessResult
VAR_INPUT
END_VAR
GetResult := stResultInternal;
END_METHOD

METHOD PUBLIC Initialise
bFlipCaptureActivePrevious := FALSE;
bFlipStart0Confirmed := FALSE;
bFlipLeft0 := FALSE;
bFlip90Seen := FALSE;
bFlipTriggerLatched := FALSE;
bFlipCaptureAccepted := FALSE;
bFlipCaptureWindowMissed := FALSE;
tonFlipDeparture(IN := FALSE);
tonTakingPictureWHileRotating(IN := FALSE);

tonStepDelay(IN := FALSE);
tonRotate180Hold(IN := FALSE);
tonMoveTimeout(IN := FALSE);



eStateInternal := E_PatchStationState.Disabled;
usiStepInternal := 0;
bHomeInternal := FALSE;
bReadyInternal := FALSE;
bBusyInternal := FALSE;
bCompleteInternal := FALSE;
bFaultInternal := FALSE;
bStopRequestInternal := FALSE;

bHorizontalBackRequestInternal := FALSE;
bHorizontalFrontRequestInternal := FALSE;
bVerticalUpRequestInternal := FALSE;
bVerticalDownRequestInternal := FALSE;

bGripCloseRequestInternal := FALSE;
bGripOpenRequestInternal := FALSE;
bRotate0RequestInternal := FALSE;
bRotate180RequestInternal := FALSE;

sDiagnosticInternal := '';

stResultInternal.bValid := FALSE;
stResultInternal.bPassed := FALSE;
stResultInternal.eCode := E_ProcessResultCode.None;
stResultInternal.udiFaultCode := 0;
stResultInternal.udiAlertCode := 0;
stResultInternal.sDetail := '';
stResultInternal.CameraResults := stEmptyVisionResults;
nVisionResultsInternal := stEmptyVisionResults;
END_METHOD

METHOD PUBLIC IsBusy : BOOL
VAR_INPUT
END_VAR
IsBusy := bBusyInternal;
END_METHOD

METHOD PUBLIC IsDone : BOOL
VAR_INPUT
END_VAR
IsDone := bCompleteInternal;
END_METHOD

METHOD PUBLIC IsFaulted : BOOL
VAR_INPUT
END_VAR
IsFaulted := bFaultInternal;
END_METHOD

METHOD PUBLIC IsReady : BOOL
VAR_INPUT
END_VAR
IsReady := bReadyInternal;
END_METHOD

METHOD PUBLIC RequestReset
VAR_INPUT
END_VAR
bFlipCaptureActivePrevious := FALSE;
bFlipStart0Confirmed := FALSE;
bFlipLeft0 := FALSE;
bFlip90Seen := FALSE;
bFlipTriggerLatched := FALSE;
bFlipCaptureAccepted := FALSE;
bFlipCaptureWindowMissed := FALSE;
tonFlipDeparture(IN := FALSE);
tonTakingPictureWHileRotating(IN := FALSE);

tonStepDelay(IN := FALSE);
tonRotate180Hold(IN := FALSE);
tonMoveTimeout(IN := FALSE);



bStopRequestInternal := FALSE;

stResultInternal.bValid := FALSE;
stResultInternal.bPassed := FALSE;
stResultInternal.eCode := E_ProcessResultCode.None;
stResultInternal.udiFaultCode := 0;
stResultInternal.udiAlertCode := 0;
stResultInternal.sDetail := '';
stResultInternal.CameraResults := stEmptyVisionResults;
nVisionResultsInternal := stEmptyVisionResults;

IF bEnableInternal AND bCommissionedInternal AND bSafetyOkInternal THEN
    IF bHomeInternal THEN
        eStateInternal := E_PatchStationState.Ready;
    ELSE
        eStateInternal := E_PatchStationState.Homing;
    END_IF
ELSE
    eStateInternal := E_PatchStationState.Disabled;
END_IF

usiStepInternal := 0;


bChangeProgramRequestInternal	:= FALSE;
bTriggerRequestInternal			:= FALSE;
bGetResultsRequestInternal		:= FALSE;
bResetResultsRequestInternal	:= FALSE;
nSetProgramNumberInternal		:= 0;
bAcknowledgeResultsInternal		:= FALSE;

bStepTargetReached 				:= FALSE;

tonTakingPictureWHileRotating.IN := FALSE;
tonCameraTriggerDelay[1].IN			:= FALSE;
tonCameraTriggerDelay[2].IN			:= FALSE;
tonDelayInspectionPlaceHolder.IN 	:= FALSE;
END_METHOD

METHOD PUBLIC RequestStart : BOOL
VAR_INPUT
END_VAR

RequestStart := FALSE;

IF bEnableInternal
    AND bCommissionedInternal
    AND bSafetyOkInternal
    AND bReadyInternal
    AND bHomeInternal
THEN
bFlipCaptureActivePrevious := FALSE;
bFlipStart0Confirmed := FALSE;
bFlipLeft0 := FALSE;
bFlip90Seen := FALSE;
bFlipTriggerLatched := FALSE;
bFlipCaptureAccepted := FALSE;
bFlipCaptureWindowMissed := FALSE;
tonFlipDeparture(IN := FALSE);
tonTakingPictureWHileRotating(IN := FALSE);

    stResultInternal.bValid := FALSE;
    stResultInternal.bPassed := FALSE;
    stResultInternal.eCode := E_ProcessResultCode.None;
    stResultInternal.udiFaultCode := 0;
    stResultInternal.udiAlertCode := 0;
    stResultInternal.sDetail := '';
    stResultInternal.CameraResults := stEmptyVisionResults;
    nVisionResultsInternal := stEmptyVisionResults;

    eStateInternal := E_PatchStationState.Processing;
    usiStepInternal := 10;
    RequestStart := TRUE;
END_IF
END_METHOD

METHOD PUBLIC RequestStop
VAR_INPUT
END_VAR
bStopRequestInternal := TRUE;
END_METHOD

METHOD PUBLIC Update
VAR_INPUT
    stProcessSettings : ST_CameraProcessSettings;
    bEnable             : BOOL;
    bCommissioned       : BOOL;
    bSafetyOk           : BOOL;
    bSupervisionEnable  : BOOL;
    bReset              : BOOL;

    // Compatibility-only inputs for removed hardware; ignored.
    bSupportRetracted   : BOOL;
    bSupportExtended    : BOOL;

    bHorizontalBack     : BOOL;
    bHorizontalFront    : BOOL;
    bVerticalUp         : BOOL;
    bVerticalDown       : BOOL;
    bLimitOff           : BOOL;
    bLimitOn            : BOOL;
    bGripOpened         : BOOL;
    bGripClosed         : BOOL;
    bRotate0            : BOOL;
    bRotate180          : BOOL;
    bRotate0Raw : BOOL;
    bRotate180Raw : BOOL;
    bCameraTriggerAccepted : BOOL;
    bCameraReadyForFlip : BOOL;
    bUseOptimizedSequenceTiming : BOOL;
	
	//CAMERA
	nCurrentProgramNumber: UDINT;
	nVisionCameraResults: ST_VisionResults;
	bResultsReady		: BOOL;

    tSupportTimeout     : TIME;
END_VAR
VAR_OUTPUT
    stStatus                 : ST_PatchStageStatus;

    bSupportExtendRequest    : BOOL;
    bSupportRetractRequest   : BOOL;
    bHorizontalBackRequest   : BOOL;
    bHorizontalFrontRequest  : BOOL;
    bVerticalUpRequest       : BOOL;
    bVerticalDownRequest     : BOOL;
    bLimitOffRequest         : BOOL;
    bLimitOnRequest          : BOOL;
    bGripCloseRequest        : BOOL;
    bGripOpenRequest         : BOOL;
    bRotate0Request          : BOOL;
    bRotate180Request        : BOOL;
	
	//camera
	bTriggerRequest			: BOOL;
	bChangeProgramRequest	: BOOL;
	bGetResultsRequest		: BOOL;
	bRequestResetResults	: BOOL;
	nProgramNumber			: UDINT;
	bAcknowledgeResults		: BOOL;

	
	
END_VAR
stProcessSettingsInternal := stProcessSettings;

	
bEnableInternal := bEnable;
bCommissionedInternal := bCommissioned;
bSafetyOkInternal := bSafetyOk;
bSupervisionEnableInternal := bSupervisionEnable;


bHorizontalBackInternal := bHorizontalBack;
bHorizontalFrontInternal := bHorizontalFront;
bVerticalUpInternal := bVerticalUp;
bVerticalDownInternal := bVerticalDown;

bGripOpenedInternal := bGripOpened;
bGripClosedInternal := bGripClosed;
bRotate0Internal := bRotate0;
bRotate180Internal := bRotate180;
bRotate0RawInternal := bRotate0Raw;
bRotate180RawInternal := bRotate180Raw;
bCameraTriggerAcceptedInternal := bCameraTriggerAccepted;
bCameraReadyForFlipInternal := bCameraReadyForFlip;
bUseOptimizedSequenceTimingInternal := bUseOptimizedSequenceTiming;


// Camera inputs must be current when reset and Cyclic evaluate the handshake.
nCurrentProgramNumberInternal	:= 		nCurrentProgramNumber;
bCameraResultsReadyInternal		:= 		bResultsReady;
nVisionResultsInternal			:= 	nVisionCameraResults;

IF bReset THEN
    RequestReset();
END_IF

Cyclic();

stStatus.eState := eStateInternal;
stStatus.bCommissioned := bCommissionedInternal;
stStatus.bHome := bHomeInternal;
stStatus.bReady := bReadyInternal;
stStatus.bBusy := bBusyInternal;
stStatus.bComplete := bCompleteInternal;
stStatus.bFault := bFaultInternal;
stStatus.eSupportFault := E_SupportCylinderFault.None; // Retired nest support.
stStatus.sDiagnostic := sDiagnosticInternal;

bSupportExtendRequest := FALSE; // Retired output, always OFF.
bSupportRetractRequest := FALSE; // Retired output, always OFF.
bHorizontalBackRequest := bHorizontalBackRequestInternal;
bHorizontalFrontRequest := bHorizontalFrontRequestInternal;
bVerticalUpRequest := bVerticalUpRequestInternal;
bVerticalDownRequest := bVerticalDownRequestInternal;
bLimitOffRequest := FALSE; // Retired output, always OFF.
bLimitOnRequest := FALSE; // Retired output, always OFF.
bGripCloseRequest := bGripCloseRequestInternal;
bGripOpenRequest := bGripOpenRequestInternal;
bRotate0Request := bRotate0RequestInternal;
bRotate180Request := bRotate180RequestInternal;

//camera
bTriggerRequest					:=		bTriggerRequestInternal;
bChangeProgramRequest			:=		bChangeProgramRequestInternal;
bGetResultsRequest				:= 		bGetResultsRequestInternal;
bRequestResetResults			:=		bResetResultsRequestInternal;
nProgramNumber 					:= 		nSetProgramNumberInternal;
bAcknowledgeResults				:= 		bAcknowledgeResultsInternal;
END_METHOD

END_FUNCTION_BLOCK

(* stored: Version 1.1.0.1, ProductVersion 3.1.4026.18
   POU FB_VisionStation: Id {da682161-7fdb-47e3-b49b-f4968c8b1f16}, SpecialFunc None
   Method Cyclic: Id {65862579-9f61-4da1-8e48-a04cc629adc5}
   Method GetResult: Id {7bfc6964-8b28-4f8c-8568-3f1997d1b2ca}
   Method Initialise: Id {b60352d8-fc31-480d-8c87-753db464b955}
   Method IsBusy: Id {6b8107df-1d67-4933-b0f5-867eee51379e}
   Method IsDone: Id {463ff2bb-de2f-4777-9e7f-15ce22a41f36}
   Method IsFaulted: Id {02d98b44-e482-4a3a-a664-c71e4343e0af}
   Method IsReady: Id {f1d3b7b6-df6d-491f-8e1a-6d304eece17e}
   Method RequestReset: Id {849d3e61-29bd-4d8e-807b-09a357055065}
   Method RequestStart: Id {a1f1fc65-484d-43e4-b289-6715c8e6c817}
   Method RequestStop: Id {c0843154-582c-4b39-b05f-d6fcabc70c1d}
   Method Update: Id {632cb56e-471f-4b5a-b14f-7c50434086c7} *)
